TYPE ZDataRecipe :
STRUCT
  RecipeParam1 : LREAL;
  RecipeParam2 : LREAL;
  RecipeParam3 : LREAL;
END_STRUCT
END_TYPE

(* stored: Version 1.1.0.1
   DUT ZDataRecipe: Id {526446ae-77f8-42f4-a19c-1ab355ad5358} *)
